{attribute 'qualified_only'}
VAR_GLOBAL CONSTANT
	analogOutputMaxVolt		: INT := 10;
	intMaxValue				: INT := 32767;
	samplingTime			: TIME := T#10S;
END_VAR

(* stored: Version 1.1.0.1, ProductVersion 3.1.4024.9
   GVL GVL_CONST: Id {e609a9ee-cdf9-4001-a1f3-11ba529f4908} *)
